INTERFACE I_Division EXTENDS I_Operator

METHOD DivideBy : I_Division
VAR_INPUT
	ipObject : I_Object;
END_VAR
VAR_OUTPUT
	e : E_OperatorError;
END_VAR
END_METHOD

END_INTERFACE

(* stored: Version 1.1.0.1, ProductVersion 3.1.4024.12
   Itf I_Division: Id {1f784833-fa93-48e6-a851-050ec3d60265}
   Method DivideBy: Id {769c7afd-a9e0-4648-bb6d-3329865fb9e0} *)
